INTERFACE I_Objekt_Kraftsensor

PROPERTY P_Messdaten : Kraftvariablen
GET
END_GET
END_PROPERTY

PROPERTY P_State : eObjectSensorState
GET
END_GET
END_PROPERTY

END_INTERFACE

(* stored: Version 1.1.0.1
   Itf I_Objekt_Kraftsensor: Id {34c6d966-f690-48ba-a1bd-ed1894f12a35}
   Property P_Messdaten: Id {ddcec799-a659-4273-8a13-41d51747c2b1}
   Get Get: Id {2cd84dd6-ace6-4b1c-8cd0-e0aeae67ed50}
   Property P_State: Id {6fb96125-7fe6-4bc6-93c4-01a8fd74fab8}
   Get Get: Id {ca6cf9e5-23e5-4cc0-9dd6-a1654dbf9690} *)
